// TwinCAT 3 PLC project PLC_SVLS_MOTION
// ProgramVersion: 3.1.4023.0
// libraries:
//   LCLS General, * (SLAC)
//   lcls-twincat-motion, * (SLAC)
//   PMPS, * (SLAC - LCLS)
//   Tc2_Standard, * (Beckhoff Automation GmbH)
//   Tc2_System, * (Beckhoff Automation GmbH)
//   Tc3_Module, * (Beckhoff Automation GmbH)
// project tree:
//   GVLs/ MAIN.TcGVL
//   / PlcTask.TcTTO
//   POUs/ PRG_ALL.TcPOU
// real-time tasks:
//   TASK PlcTask: cycle T#10ms, priority 20, ADS port 350
// motion (NC):
//   TASK SVLS_MOTION SAF: cycle T#2ms, priority 4, ADS port 501
//   TASK SVLS_MOTION SVB: cycle T#10ms, priority 8, ADS port 511
//   AXIS M1_DET_Y (id 1)
//     General: UnitName=Degree
//     Dynamic: AccelerationMaximum=0.572958, DecelerationMaximum=0.572958
//     Velo: Maximum=0.02
//     OtherSettings: AllowMotionCmdToSlave=true
//     encoder EncType=29
//       EncPara: ScaleFactorNumerator=8.3819032e-08, MaxCount=#xffffffff, MaxCountHighDWord=#x0000001f
//         Inc: RefSoftSyncMask=#x0000ffff
//     drive DrvType=24
//       Analog: VeloReferenz=0.025492, TorqueSetpointScale=10, ScaleFactorActTorque=0.1
//       TimeComp: TaskDelayCycles=1
//     controller CtrType=1
//       CtrPara: PriorControlFactor=1
//         PosDiffControl: Range=0.6
//         Observer: BandWidth=20
//   AXIS M2_DET_Z (id 2)
//     Dynamic: AccelerationMaximum=50, DecelerationMaximum=50, Acceleration=50, Deceleration=50
//     Velo: RefSearch=0.1, RefSync=0.1, SlowManual=0.25, FastManual=0.5, Maximum=0.5
//     TargetPosControl: Range=0.01
//     OtherSettings: AllowMotionCmdToSlave=true
//     encoder EncType=29
//       EncPara: ScaleFactorNumerator=5e-05, Offset=-6871872.3264, MaxCount=#xffffffff, MaxCountHighDWord=#x0000001f
//         SoftEndMinControl: Enable=true, Range=-53.8
//         SoftEndMaxControl: Enable=true, Range=51.3
//         Inc: RefSoftSyncMask=#x0000ffff
//     drive DrvType=24
//       Analog: VeloReferenz=0.5, TorqueSetpointScale=10, ScaleFactorActTorque=0.1
//       TimeComp: TaskDelayCycles=1
//     controller CtrType=1
//       CtrPara: PriorControlFactor=1
//         PosDiffControl: Range=0.07
//         Observer: BandWidth=20
//   AXIS M3_GRA_Y (id 3)
//     Dynamic: AccelerationMaximum=5, DecelerationMaximum=5, Acceleration=5, Deceleration=5, Jerk=5
//     Velo: RefSearch=0.01, RefSync=0.01, SlowManual=0.0025, FastManual=0.005, Maximum=0.05
//     PositionAreaControl: Range=0.003
//     TargetPosControl: Range=0.0002
//     OtherSettings: AllowMotionCmdToSlave=true
//     encoder EncType=29
//       EncPara: ScaleFactorNumerator=5e-05, Offset=-17.0296, MaxCount=#xffffffff, MaxCountHighDWord=#x0000001f
//         SoftEndMinControl: Enable=true, Range=-1.11
//         SoftEndMaxControl: Enable=true, Range=1.35
//         Inc: RefSoftSyncMask=#x0000ffff
//     drive DrvType=24
//       DrvPara: Inverse=true
//         Analog: VeloReferenz=0.106, TorqueSetpointScale=10, ScaleFactorActTorque=0.1
//         TimeComp: TaskDelayCycles=1
//     controller CtrType=1
//       CtrPara: PriorControlFactor=1
//         PosDiffControl: Range=0.1
//         Observer: BandWidth=20
//   AXIS M4_SLITX_L (id 4)
//     OtherSettings: AllowMotionCmdToSlave=true
//     encoder EncType=29
//       EncPara: ScaleFactorNumerator=5e-05, MaxCount=#xffffffff, MaxCountHighDWord=#x0000001f, ReferenceSystem=1
//     drive DrvType=5
//       Analog: TorqueSetpointScale=10, ScaleFactorActTorque=0.1
//       TimeComp: TaskDelayCycles=1
//     controller CtrType=1
//       CtrPara: PriorControlFactor=1
//         Observer: BandWidth=20
//   AXIS M5_SLITX_R (id 5)
//     OtherSettings: AllowMotionCmdToSlave=true
//     encoder EncType=29
//       EncPara: ScaleFactorNumerator=5e-05, MaxCount=#xffffffff, MaxCountHighDWord=#x0000001f
//     drive DrvType=5
//       Analog: TorqueSetpointScale=10, ScaleFactorActTorque=0.1
//       TimeComp: TaskDelayCycles=1
//     controller CtrType=1
//       CtrPara: PriorControlFactor=1
//         Observer: BandWidth=20
//   AXIS M6_SLITY_T (id 6)
//     OtherSettings: AllowMotionCmdToSlave=true
//     encoder EncType=29
//       EncPara: ScaleFactorNumerator=5e-05, MaxCount=#xffffffff, MaxCountHighDWord=#x0000001f
//     drive DrvType=5
//       Analog: TorqueSetpointScale=10, ScaleFactorActTorque=0.1
//       TimeComp: TaskDelayCycles=1
//     controller CtrType=1
//       CtrPara: PriorControlFactor=1
//         Observer: BandWidth=20
//   AXIS M7_SLITY_B (id 7)
//     OtherSettings: AllowMotionCmdToSlave=true
//     encoder EncType=29
//       EncPara: ScaleFactorNumerator=5e-05, MaxCount=#xffffffff, MaxCountHighDWord=#x0000001f, ReferenceSystem=1
//     drive DrvType=5
//       Analog: TorqueSetpointScale=10, ScaleFactorActTorque=0.1
//       TimeComp: TaskDelayCycles=1
//     controller CtrType=1
//       CtrPara: PriorControlFactor=1
//         Observer: BandWidth=20
// I/O:
//   DEVICE Device 1 (EtherCAT), AmsNetId 199.4.42.250.2.1
//     EK1200_01_00 [EK1200-5000 EtherCAT Power supply (2A E-Bus)]
//       EL6070_01_00 [EL6070 1Ch. Licensing-Terminal]
//       EL7047_01_01-DET_Y [EL7047 1Ch. Stepper motor output stage (50V, 5A)]
//       EL5042_01_02-DET_Y-DET_Z [EL5042 2Ch. BiSS-C Encoder]
//       EL7047_01_03-DET_Z [EL7047 1Ch. Stepper motor output stage (50V, 5A)]
//       EL7047_01_04-GRT_Y [EL7047 1Ch. Stepper motor output stage (50V, 5A)]
//       EL5042_01_05-GRT_Y-SP5 [EL5042 2Ch. BiSS-C Encoder]
//       EL5042_01_06-SP1-SP2 [EL5042 2Ch. BiSS-C Encoder]
//       EL5042_01_07-SP3-SP4 [EL5042 2Ch. BiSS-C Encoder]
//       EL9011_01_Endstop [EL9011 End Terminal]
// variable links:
//   (this object) <-> Device 1 (EtherCAT)/Term 1 (EK1100)/EL5042_00_03
//     Enc/Inputs/In/nComState @bit 1 <-> WcState/InputToggle
//     Enc/Inputs/In/nComState <-> WcState/WcState
//     Enc/Inputs/In/nDataIn1 <-> FB Inputs Channel 1/Position
//     Enc/Inputs/In/nState1 @bit 12 <-> FB Inputs Channel 1/Status/Diag
//     Enc/Inputs/In/nState1 @bit 1 <-> FB Inputs Channel 1/Status/Error
//     Enc/Inputs/In/nState1 @bit 14 <-> FB Inputs Channel 1/Status/Input cycle counter
//     Enc/Inputs/In/nState1 @bit 2 <-> FB Inputs Channel 1/Status/Ready
//     Enc/Inputs/In/nState1 @bit 13 <-> FB Inputs Channel 1/Status/TxPDO State
//     Enc/Inputs/In/nState1 <-> FB Inputs Channel 1/Status/Warning
//   (this object) <-> Device 1 (EtherCAT)/Term 1 (EK1100)/EL7047_00_02
//     Drive/Inputs/In/nState1 @bit 3 <-> STM Status/Status/Error
//     Drive/Inputs/In/nState1 @bit 7 <-> STM Status/Status/Motor stall
//     Drive/Inputs/In/nState1 @bit 5 <-> STM Status/Status/Moving negative
//     Drive/Inputs/In/nState1 @bit 4 <-> STM Status/Status/Moving positive
//     Drive/Inputs/In/nState1 @bit 1 <-> STM Status/Status/Ready
//     Drive/Inputs/In/nState1 <-> STM Status/Status/Ready to enable
//     Drive/Inputs/In/nState1 @bit 6 <-> STM Status/Status/Torque reduced
//     Drive/Inputs/In/nState1 @bit 2 <-> STM Status/Status/Warning
//     Drive/Inputs/In/nState2 @bit 3 <-> STM Status/Status/Digital input 1
//     Drive/Inputs/In/nState2 @bit 4 <-> STM Status/Status/Digital input 2
//     Drive/Inputs/In/nState2 @bit 5 <-> STM Status/Status/Sync error
//     Drive/Inputs/In/nState2 @bit 7 <-> STM Status/Status/TxPDO Toggle
//     Drive/Inputs/In/nState4 @bit 1 <-> WcState/InputToggle
//     Drive/Inputs/In/nState4 <-> WcState/WcState
//     Drive/Outputs/Out/nCtrl1 <-> STM Control/Control/Enable
//     Drive/Outputs/Out/nCtrl1 @bit 2 <-> STM Control/Control/Reduce torque
//     Drive/Outputs/Out/nCtrl1 @bit 1 <-> STM Control/Control/Reset
//     Drive/Outputs/Out/nCtrl2 @bit 3 <-> STM Control/Control/Digital output 1
//     Drive/Outputs/Out/nDataOut2[0] <-> STM Velocity/Velocity
//   (this object) <-> Device 1 (EtherCAT)/EK1200_01_00/EL5042_01_02-DET_Y-DET_Z
//     Enc/Inputs/In/nComState @bit 1 <-> WcState/InputToggle
//     Enc/Inputs/In/nComState <-> WcState/WcState
//     Enc/Inputs/In/nDataIn1 <-> FB Inputs Channel 2/Position
//     Enc/Inputs/In/nState1 @bit 12 <-> FB Inputs Channel 2/Status/Diag
//     Enc/Inputs/In/nState1 @bit 1 <-> FB Inputs Channel 2/Status/Error
//     Enc/Inputs/In/nState1 @bit 14 <-> FB Inputs Channel 2/Status/Input cycle counter
//     Enc/Inputs/In/nState1 @bit 2 <-> FB Inputs Channel 2/Status/Ready
//     Enc/Inputs/In/nState1 @bit 13 <-> FB Inputs Channel 2/Status/TxPDO State
//     Enc/Inputs/In/nState1 <-> FB Inputs Channel 2/Status/Warning
//   (this object) <-> Device 1 (EtherCAT)/EK1200_01_00/EL7047_01_03-DET_Z
//     Drive/Inputs/In/nState1 @bit 3 <-> STM Status/Status/Error
//     Drive/Inputs/In/nState1 @bit 7 <-> STM Status/Status/Motor stall
//     Drive/Inputs/In/nState1 @bit 5 <-> STM Status/Status/Moving negative
//     Drive/Inputs/In/nState1 @bit 4 <-> STM Status/Status/Moving positive
//     Drive/Inputs/In/nState1 @bit 1 <-> STM Status/Status/Ready
//     Drive/Inputs/In/nState1 <-> STM Status/Status/Ready to enable
//     Drive/Inputs/In/nState1 @bit 6 <-> STM Status/Status/Torque reduced
//     Drive/Inputs/In/nState1 @bit 2 <-> STM Status/Status/Warning
//     Drive/Inputs/In/nState2 @bit 3 <-> STM Status/Status/Digital input 1
//     Drive/Inputs/In/nState2 @bit 4 <-> STM Status/Status/Digital input 2
//     Drive/Inputs/In/nState2 @bit 5 <-> STM Status/Status/Sync error
//     Drive/Inputs/In/nState2 @bit 7 <-> STM Status/Status/TxPDO Toggle
//     Drive/Inputs/In/nState4 @bit 1 <-> WcState/InputToggle
//     Drive/Inputs/In/nState4 <-> WcState/WcState
//     Drive/Outputs/Out/nCtrl1 <-> STM Control/Control/Enable
//     Drive/Outputs/Out/nCtrl1 @bit 2 <-> STM Control/Control/Reduce torque
//     Drive/Outputs/Out/nCtrl1 @bit 1 <-> STM Control/Control/Reset
//     Drive/Outputs/Out/nCtrl2 @bit 3 <-> STM Control/Control/Digital output 1
//     Drive/Outputs/Out/nDataOut2[0] <-> STM Velocity/Velocity
//   (this object) <-> Device 1 (EtherCAT)/EK1200_01_00/EL5042_01_05-GRT_Y-SP5
//     Enc/Inputs/In/nComState @bit 1 <-> WcState/InputToggle
//     Enc/Inputs/In/nComState <-> WcState/WcState
//     Enc/Inputs/In/nDataIn1 <-> FB Inputs Channel 1/Position
//     Enc/Inputs/In/nState1 @bit 12 <-> FB Inputs Channel 1/Status/Diag
//     Enc/Inputs/In/nState1 @bit 1 <-> FB Inputs Channel 1/Status/Error
//     Enc/Inputs/In/nState1 @bit 14 <-> FB Inputs Channel 1/Status/Input cycle counter
//     Enc/Inputs/In/nState1 @bit 2 <-> FB Inputs Channel 1/Status/Ready
//     Enc/Inputs/In/nState1 @bit 13 <-> FB Inputs Channel 1/Status/TxPDO State
//     Enc/Inputs/In/nState1 <-> FB Inputs Channel 1/Status/Warning
//   (this object) <-> Device 1 (EtherCAT)/EK1200_01_00/EL7047_01_04-GRT_Y
//     Drive/Inputs/In/nState1 @bit 3 <-> STM Status/Status/Error
//     Drive/Inputs/In/nState1 @bit 7 <-> STM Status/Status/Motor stall
//     Drive/Inputs/In/nState1 @bit 5 <-> STM Status/Status/Moving negative
//     Drive/Inputs/In/nState1 @bit 4 <-> STM Status/Status/Moving positive
//     Drive/Inputs/In/nState1 @bit 1 <-> STM Status/Status/Ready
//     Drive/Inputs/In/nState1 <-> STM Status/Status/Ready to enable
//     Drive/Inputs/In/nState1 @bit 6 <-> STM Status/Status/Torque reduced
//     Drive/Inputs/In/nState1 @bit 2 <-> STM Status/Status/Warning
//     Drive/Inputs/In/nState2 @bit 3 <-> STM Status/Status/Digital input 1
//     Drive/Inputs/In/nState2 @bit 4 <-> STM Status/Status/Digital input 2
//     Drive/Inputs/In/nState2 @bit 5 <-> STM Status/Status/Sync error
//     Drive/Inputs/In/nState2 @bit 7 <-> STM Status/Status/TxPDO Toggle
//     Drive/Inputs/In/nState4 @bit 1 <-> WcState/InputToggle
//     Drive/Inputs/In/nState4 <-> WcState/WcState
//     Drive/Outputs/Out/nCtrl1 <-> STM Control/Control/Enable
//     Drive/Outputs/Out/nCtrl1 @bit 2 <-> STM Control/Control/Reduce torque
//     Drive/Outputs/Out/nCtrl1 @bit 1 <-> STM Control/Control/Reset
//     Drive/Outputs/Out/nCtrl2 @bit 3 <-> STM Control/Control/Digital output 1
//     Drive/Outputs/Out/nDataOut2[0] <-> STM Velocity/Velocity
//   (this object) <-> Device 1 (EtherCAT)/Term 1 (EK1100)/EL5042_00_07
//     Enc/Inputs/In/nComState @bit 1 <-> WcState/InputToggle
//     Enc/Inputs/In/nComState <-> WcState/WcState
//     Enc/Inputs/In/nDataIn1 <-> FB Inputs Channel 2/Position
//     Enc/Inputs/In/nState1 @bit 12 <-> FB Inputs Channel 2/Status/Diag
//     Enc/Inputs/In/nState1 @bit 1 <-> FB Inputs Channel 2/Status/Error
//     Enc/Inputs/In/nState1 @bit 14 <-> FB Inputs Channel 2/Status/Input cycle counter
//     Enc/Inputs/In/nState1 @bit 2 <-> FB Inputs Channel 2/Status/Ready
//     Enc/Inputs/In/nState1 @bit 13 <-> FB Inputs Channel 2/Status/TxPDO State
//     Enc/Inputs/In/nState1 <-> FB Inputs Channel 2/Status/Warning
//   (this object) <-> Device 1 (EtherCAT)/Term 1 (EK1100)/EL5042_00_08
//     Enc/Inputs/In/nComState @bit 1 <-> WcState/InputToggle
//     Enc/Inputs/In/nComState <-> WcState/WcState
//     Enc/Inputs/In/nDataIn1 <-> FB Inputs Channel 1/Position
//     Enc/Inputs/In/nState1 @bit 12 <-> FB Inputs Channel 1/Status/Diag
//     Enc/Inputs/In/nState1 @bit 1 <-> FB Inputs Channel 1/Status/Error
//     Enc/Inputs/In/nState1 @bit 14 <-> FB Inputs Channel 1/Status/Input cycle counter
//     Enc/Inputs/In/nState1 @bit 2 <-> FB Inputs Channel 1/Status/Ready
//     Enc/Inputs/In/nState1 @bit 13 <-> FB Inputs Channel 1/Status/TxPDO State
//     Enc/Inputs/In/nState1 <-> FB Inputs Channel 1/Status/Warning
//   PLC_SVLS_MOTION Instance <-> Device 1 (EtherCAT)/Term 1 (EK1100)/EL5042_00_03
//     PlcTask Inputs/MAIN.M1.nRawEncoderULINT <-> FB Inputs Channel 1/Position
//     PlcTask Inputs/MAIN.M2.nRawEncoderULINT <-> FB Inputs Channel 2/Position
//   PLC_SVLS_MOTION Instance <-> Device 1 (EtherCAT)/Term 1 (EK1100)/EL5042_00_06
//     PlcTask Inputs/MAIN.M3.nRawEncoderULINT <-> FB Inputs Channel 1/Position
//   PLC_SVLS_MOTION Instance <-> Device 1 (EtherCAT)/Term 1 (EK1100)/EL5042_00_07
//     PlcTask Inputs/MAIN.ENC_X_L.nRawEncoderULINT <-> FB Inputs Channel 1/Position
//     PlcTask Inputs/MAIN.ENC_X_R.nRawEncoderULINT <-> FB Inputs Channel 1/Position
//     PlcTask Inputs/MAIN.ENC_Y_B.nRawEncoderULINT <-> FB Inputs Channel 1/Position
//     PlcTask Inputs/MAIN.ENC_Y_T.nRawEncoderULINT <-> FB Inputs Channel 1/Position
//   PLC_SVLS_MOTION Instance <-> Device 1 (EtherCAT)/Term 1 (EK1100)/EL7047_00_02
//     PlcTask Inputs/MAIN.M1.bLimitBackwardEnable <-> STM Status/Status/Digital input 2
//     PlcTask Inputs/MAIN.M1.bLimitForwardEnable <-> STM Status/Status/Digital input 1
//   PLC_SVLS_MOTION Instance <-> Device 1 (EtherCAT)/Term 1 (EK1100)/EL7047_00_04
//     PlcTask Inputs/MAIN.M2.bLimitBackwardEnable <-> STM Status/Status/Digital input 2
//     PlcTask Inputs/MAIN.M2.bLimitForwardEnable <-> STM Status/Status/Digital input 1
//   PLC_SVLS_MOTION Instance <-> Device 1 (EtherCAT)/Term 1 (EK1100)/EL7047_00_05
//     PlcTask Inputs/MAIN.M3.bLimitBackwardEnable <-> STM Status/Status/Digital input 2
//     PlcTask Inputs/MAIN.M3.bLimitForwardEnable <-> STM Status/Status/Digital input 1
//   PLC_SVLS_MOTION Instance <-> SVLS_MOTION SAF/Axes/M1_DET_Y
//     PlcTask Inputs/MAIN.M1.Axis.NcToPlc <-> Outputs/ToPlc
//     PlcTask Outputs/MAIN.M1.Axis.PlcToNc <-> Inputs/FromPlc
//   PLC_SVLS_MOTION Instance <-> SVLS_MOTION SAF/Axes/M2_DET_Z
//     PlcTask Inputs/MAIN.M2.Axis.NcToPlc <-> Outputs/ToPlc
//     PlcTask Outputs/MAIN.M2.Axis.PlcToNc <-> Inputs/FromPlc
//   PLC_SVLS_MOTION Instance <-> SVLS_MOTION SAF/Axes/M3_GRA_Y
//     PlcTask Inputs/MAIN.M3.Axis.NcToPlc <-> Outputs/ToPlc
//     PlcTask Outputs/MAIN.M3.Axis.PlcToNc <-> Inputs/FromPlc
//   PLC_SVLS_MOTION Instance <-> SVLS_MOTION SAF/Axes/M4_SLITX_L
//     PlcTask Inputs/MAIN.ENC_X_L.Axis.NcToPlc <-> Outputs/ToPlc
//     PlcTask Outputs/MAIN.ENC_X_L.Axis.PlcToNc <-> Inputs/FromPlc
//   PLC_SVLS_MOTION Instance <-> SVLS_MOTION SAF/Axes/M5_SLITX_R
//     PlcTask Inputs/MAIN.ENC_X_R.Axis.NcToPlc <-> Outputs/ToPlc
//     PlcTask Outputs/MAIN.ENC_X_R.Axis.PlcToNc <-> Inputs/FromPlc
//   PLC_SVLS_MOTION Instance <-> SVLS_MOTION SAF/Axes/M6_SLITY_T
//     PlcTask Inputs/MAIN.ENC_Y_T.Axis.NcToPlc <-> Outputs/ToPlc
//     PlcTask Outputs/MAIN.ENC_Y_T.Axis.PlcToNc <-> Inputs/FromPlc
//   PLC_SVLS_MOTION Instance <-> SVLS_MOTION SAF/Axes/M7_SLITY_B
//     PlcTask Inputs/MAIN.ENC_Y_B.Axis.NcToPlc <-> Outputs/ToPlc
//     PlcTask Outputs/MAIN.ENC_Y_B.Axis.PlcToNc <-> Inputs/FromPlc

CONFIGURATION PLC_SVLS_MOTION
    RESOURCE PLC ON TwinCAT3
        TASK PlcTask(INTERVAL := T#10ms, PRIORITY := 20);
        PROGRAM PRG_ALL WITH PlcTask : PRG_ALL;
    END_RESOURCE
END_CONFIGURATION

// ---- GVLs/MAIN.TcGVL
{attribute 'qualified_only'}
VAR_GLOBAL
    {attribute 'pytmc' := 'pv: CRIXS:SVLS:DET:MMS:Y'}
    {attribute 'TcLinkTo' := '.bLimitForwardEnable  := TIIB[EL7047_00_02]^STM Status^Status^Digital input 1;
                              .bLimitBackwardEnable := TIIB[EL7047_00_02]^STM Status^Status^Digital input 2;
                              .nRawEncoderULINT     := TIIB[EL5042_00_03]^FB Inputs Channel 1^Position'}
    M1: ST_MotionStage := (sName := 'CRIXS:SVLS:DET:MMS:Y');

    {attribute 'pytmc' := 'pv: CRIXS:SVLS:DET:MMS:Z'}
    {attribute 'TcLinkTo' := '.bLimitForwardEnable  := TIIB[EL7047_00_04]^STM Status^Status^Digital input 1;
                              .bLimitBackwardEnable := TIIB[EL7047_00_04]^STM Status^Status^Digital input 2;
                              .nRawEncoderULINT     := TIIB[EL5042_00_03]^FB Inputs Channel 2^Position'}
    M2: ST_MotionStage := (sName := 'CRIXS:SVLS:DET:MMS:Z');

    {attribute 'pytmc' := 'pv: CRIXS:SVLS:GRA:MMS:Y'}
    {attribute 'TcLinkTo' := '.bLimitForwardEnable  := TIIB[EL7047_00_05]^STM Status^Status^Digital input 1;
                              .bLimitBackwardEnable := TIIB[EL7047_00_05]^STM Status^Status^Digital input 2;
                              .nRawEncoderULINT     := TIIB[EL5042_00_06]^FB Inputs Channel 1^Position'}
    M3: ST_MotionStage := (sName := 'CRIXS:SVLS:GRA:MMS:Y');

///Encoder linking for SmarACT stages
//SLITS X
    {attribute 'pytmc' := 'pv:	CRIXS:SVLS:SLITSX:ENC:L'}
    {attribute 'TcLinkTo' := '.nRawEncoderULINT     := TIIB[EL5042_00_07]^FB Inputs Channel 1^Position;'}
    ENC_X_L : ST_MotionStage := (sName := 'CRIXS:SVLS:SLITSX:ENC:L');

    {attribute 'pytmc' := 'pv:	CRIXS:SVLS:SLITSX:ENC:R'}
    {attribute 'TcLinkTo' := '.nRawEncoderULINT     := TIIB[EL5042_00_07]^FB Inputs Channel 1^Position;'}
    ENC_X_R : ST_MotionStage := (sName := 'CRIXS:SVLS:SLITSX:ENC:R');
//SLITS Y
    {attribute 'pytmc' := 'pv:	CRIXS:SVLS:SLITSY:ENC:T'}
    {attribute 'TcLinkTo' := '.nRawEncoderULINT     := TIIB[EL5042_00_07]^FB Inputs Channel 1^Position;'}
    ENC_Y_T : ST_MotionStage := (sName := 'CRIXS:SVLS:SLITSY:ENC:T');

    {attribute 'pytmc' := 'pv:	CRIXS:SVLS:SLITSY:ENC:B'}
    {attribute 'TcLinkTo' := '.nRawEncoderULINT     := TIIB[EL5042_00_07]^FB Inputs Channel 1^Position;'}
    ENC_Y_B : ST_MotionStage := (sName := 'CRIXS:SVLS:SLITSY:ENC:B');

END_VAR

// ---- POUs/PRG_ALL.TcPOU
PROGRAM PRG_ALL
VAR
    fb_DET_Y : FB_MotionStage;
    fb_DET_Z : FB_MotionStage;
    fb_GRA_Y : FB_MotionStage;
    bInit : BOOl := TRUE;
END_VAR

IF ( bInit) THEN
    bInit := FALSE;
    Main.M1.bHardwareEnable := TRUE;
    Main.M1.bPowerSelf := TRUE;
    Main.M1.nBrakeMode := ENUM_StageBrakeMode.NO_BRAKE;
    Main.M1.nEnableMode := ENUM_StageEnableMode.DURING_MOTION;

    Main.M2.bHardwareEnable := TRUE;
    Main.M2.bPowerSelf := TRUE;
    Main.M2.nBrakeMode := ENUM_StageBrakeMode.NO_BRAKE;
    Main.M2.nEnableMode := ENUM_StageEnableMode.DURING_MOTION;

    Main.M3.bHardwareEnable := TRUE;
    Main.M3.bPowerSelf := TRUE;
    Main.M3.nBrakeMode := ENUM_StageBrakeMode.NO_BRAKE;
    Main.M3.nEnableMode := ENUM_StageEnableMode.DURING_MOTION;

END_IF

fb_DET_Y(stMotionStage:=Main.M1);
fb_DET_Z(stMotionStage:=Main.M2);
fb_GRA_Y(stMotionStage:=Main.M3);

END_PROGRAM
